// TIA Portal V19 export
FUNCTION_BLOCK "TYPIC_C106_IF_HSI"   // FB99, FBD
TITLE = TYPIC_C106_IF_HSI: Hoogspanningsinstallatie
{ S7_Optimized_Access := 'TRUE' }
AUTHOR : OCOTECH
FAMILY : Typical
NAME : C106.701
// Logisch Object Besturing: C106.701
// 
// De interne functie Hoogspanningsinstallatie verzorgt de bewaking van een hoogspanningsinstallatie.
// stored: MemoryReserve 10, SetENOAutomatically false
   VAR_INPUT
      EXT_AUT { ExternalAccessible := 'False'; ExternalVisible := 'False'; ExternalWritable := 'False'} : Bool;   // Externe (hoofd) beveiliging (1 = OK)
      EXT_HW { ExternalAccessible := 'False'; ExternalVisible := 'False'; ExternalWritable := 'False'} : Bool;   // Sturings hardware (PLC) bewaking (1 = OK)
      IN_STO_NOK { ExternalAccessible := 'False'; ExternalVisible := 'False'; ExternalWritable := 'False'} : Bool;   // Storing aanwezig die niet observeerbaar tot gevolg heeft
      IN_STO_OK { ExternalAccessible := 'False'; ExternalVisible := 'False'; ExternalWritable := 'False'} : Bool;   // Storing aanwezig die observeerbaarheid niet beinvloed
      IN_HSI_BSC1 { ExternalAccessible := 'False'; ExternalVisible := 'False'; ExternalWritable := 'False'} : Bool;   // Hoogspanningsinstallatie beschikbaar
      IN_HSI_BSC2 { ExternalAccessible := 'False'; ExternalVisible := 'False'; ExternalWritable := 'False'} : Bool;   // Hoogspanningsinstallatie niet beschikbaar
      IN_HSI_BSC3 { ExternalAccessible := 'False'; ExternalVisible := 'False'; ExternalWritable := 'False'} : Bool;   // Hoogspanningsinstallatie beperkt beschikbaar
      IN_LUS_TOE { ExternalAccessible := 'False'; ExternalVisible := 'False'; ExternalWritable := 'False'} : Bool;   // Hoogspanningslus is gesloten
      IN_WRE1 { ExternalAccessible := 'False'; ExternalVisible := 'False'; ExternalWritable := 'False'} : Bool;   // Werkingsregime: Netbedrijf
      IN_WRE2 { ExternalAccessible := 'False'; ExternalVisible := 'False'; ExternalWritable := 'False'} : Bool;   // Werkingsregime: Parallelbedrijf
      IN_WRE3 { ExternalAccessible := 'False'; ExternalVisible := 'False'; ExternalWritable := 'False'} : Bool;   // Werkingsregime: Eilandbedrijf
      IN_HSI_ENE_TOT { ExternalAccessible := 'False'; ExternalVisible := 'False'; ExternalWritable := 'False'} : Real;   // Totaal energieverbruik hoogspanningsinstallatie
      IN_AUT_C106 { ExternalAccessible := 'False'; ExternalVisible := 'False'; ExternalWritable := 'False'} : Bool;   // Beveiligingen: serie geschakelde terugmelding (1 = OK)
   END_VAR
   VAR_OUTPUT
      VAR_IF_HSI { ExternalAccessible := 'False'; ExternalVisible := 'False'; ExternalWritable := 'False'} : "C106_VAR_IF_HSI_TYPIC";   // Struct met alle variabelen naar bovenliggende functies
   END_VAR
   VAR
      STO { ExternalWritable := 'False'} : Struct   // Storingen
         A001 : Bool;   // Beveiliging aangesproken
         A002 : Bool;   // Hoogspanningsinstallatie in storing
         A003 : Bool;   // Algemene storing hoogspanningsinstallatie
         A004 : Bool;   // Hoogspanningslus is geopend
      END_STRUCT;
      VAR { ExternalWritable := 'False'} : Struct   // Variabelen
         BSC1 : Bool;   // Hoogspanningsinstallatie beschikbaar
         BSC2 : Bool;   // Hoogspanningsinstallatie niet beschikbaar
         BSC3 : Bool;   // Hoogspanningsinstallatie beperkt beschikbaar
         WRE1 : Bool;   // Werkingsregime: Netbedrijf
         WRE2 : Bool;   // Werkingsregime: Parallelbedrijf
         WRE3 : Bool;   // Werkingsregime: Eilandbedrijf
         LUS_TOE : Bool;   // Hoogspanningslus is gesloten
         EXT_AUT { ExternalAccessible := 'False'; ExternalVisible := 'False'} : Bool;   // Externe (hoofd) beveiliging aangesproken
         EXT_HW { ExternalAccessible := 'False'; ExternalVisible := 'False'} : Bool;   // Sturings hardware (PLC) in storing
      END_STRUCT;
   END_VAR
BEGIN

REGION Network 1: START
END_REGION

REGION Network 2: +++ Verwerking meetwaarden en statussen +++
   // De meetwaarde en status wordt ontvangen vanuit de interne sturing.
END_REGION

REGION Network 3: +++ Storingen +++
   // Verwerken van de storingsmeldingen (inputs).
END_REGION

REGION Network 4: Storing A001: Beveiliging aangesproken
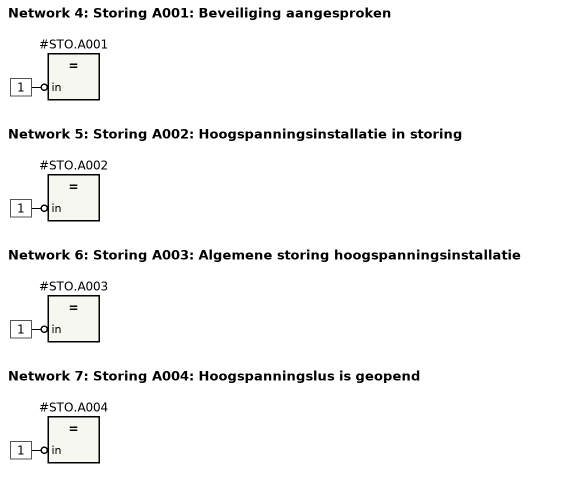
   #STO.A001 := NOT 1;
END_REGION

REGION Network 5: Storing A002: Hoogspanningsinstallatie in storing
   #STO.A002 := NOT 1;
END_REGION

REGION Network 6: Storing A003: Algemene storing hoogspanningsinstallatie
   #STO.A003 := NOT 1;
END_REGION

REGION Network 7: Storing A004: Hoogspanningslus is geopend
   #STO.A004 := NOT 1;
END_REGION

REGION Network 8 (SCL): EINDE
   // Variabelen van intern scada rakvlak naar outputs copieren
   #VAR_IF_HSI.BSC1 := #VAR.BSC1;
   #VAR_IF_HSI.BSC2 := #VAR.BSC2;
   #VAR_IF_HSI.BSC3 := #VAR.BSC3;
   #VAR_IF_HSI.WRE1 := #VAR.WRE1;
   #VAR_IF_HSI.WRE2 := #VAR.WRE2;
   #VAR_IF_HSI.WRE3 := #VAR.WRE3;
   #VAR_IF_HSI.LUS_TOE := #VAR.LUS_TOE;
   #VAR_IF_HSI.EXT_AUT := #VAR.EXT_AUT;
   #VAR_IF_HSI.EXT_HW := #VAR.EXT_HW;
   #VAR_IF_HSI.STO := #STO;
END_REGION
END_FUNCTION_BLOCK
